// TIA Portal V20 export
DATA_BLOCK "QDAS_InterfaceRelation"   // DB299
{ S7_Optimized_Access := 'TRUE' }
// stored: MemoryReserve 100
   VAR
      Q_DAS : Struct
         commands : Struct
            reset : Bool;
            trigger : Bool;
         END_STRUCT;
         monitoring : Struct
            done : Bool;
            error : Bool;
         END_STRUCT;
      END_STRUCT;
   END_VAR
BEGIN
END_DATA_BLOCK
